RoboDK station: coursework2_ReiaMenezes_M00791121_finalsubmission.rdk

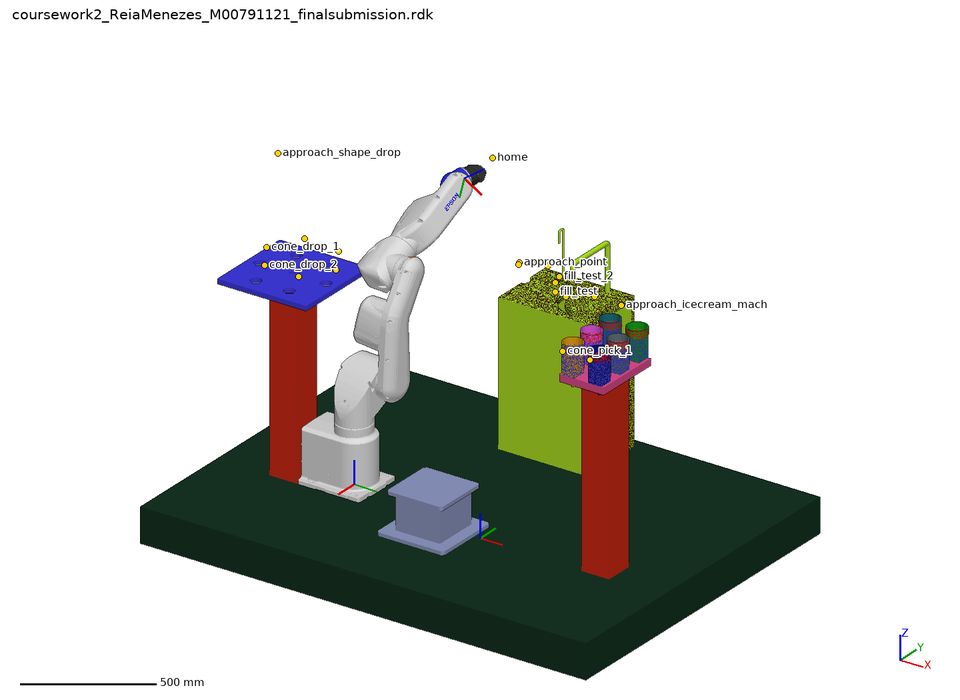
[picture v0: the station drawn from its stored meshes, robots at their saved joint values, targets as dots, program paths as lines]
Station coursework2_ReiaMenezes_M00791121_finalsubmission (saved by RoboDK 5.8.0). Poses are relative to the parent item; angles as X-Y-Z fixed-axis rotations.
Station parameters (name, value as stored): 153.91
  - frame Base_cell_frame at (0, 0, 0) mm
    - object PDE4431_CW2_2024 at (0, 0, 0) mm, rotated rx 90 ry 0 rz 0 deg, size 2000 x 980 x 1500 mm, geometry from PDE4431_CW2_2024.STEP
    - frame Epson VT6 Base at (-250, -450, 330) mm, rotated rx 0 ry 0 rz -90 deg
      - robot Epson VT6: 6 axes, payload 6 kg, reach 920 mm, repeatability 0.1 mm, weight 40 kg
          modified DH rows (alpha deg, a mm, theta deg, d mm): 0, 0, 0, 412; -90, 100, -90, 0; 0, 420, 0, 0; -90, 0, 0, 400; 90, 0, 0, 0; -90, 0, 0, 80
          base shift (0, 0, 0) mm, rotated rx 0 ry 0 rz 90 deg
          joint limits [-170, -160, -51, -200, -125, -360] to [170, 65, 190, 200, 125, 360]; home [0, 0, 0, 0, 0, 0]; saved at [85.974, -13.175, 41.561, 23.33, -25.202, -130.293]
        - frame RobotiQ 2F-140 Gripper (Mechanism) Base at (0, 0, 0) mm
          - robot RobotiQ 2F-140 Gripper (Mechanism) (model RobotiQ 2F140): 1 axes, payload 5 kg
              joint limits [0] to [140]; home [140]; saved at [99.47]
          - target open_gripper (Cartesian target) at (0, 0, 135) mm, rotated rx -90 ry 0 rz 90 deg; joints [99.47, 14.65, 163.72, -0.95, 89.45, -5.12] of RobotiQ 2F-140 Gripper (Mechanism)
          - target close_gripper (Cartesian target) at (0, 0, 135) mm, rotated rx -90 ry 0 rz 90 deg; joints [60, 27.47, -32.86, -122.29, -24.8, -148.93] of RobotiQ 2F-140 Gripper (Mechanism)
        - tool Tool 1, TCP at (-20, -10, 155) mm, rotated rx -100 ry 0 rz 70 deg
    - object Pedestal_1 at (0, -300, 150) mm, rotated rx 90 ry 0 rz 0 deg, size 300 x 180 x 300 mm, geometry from Pedestal_1.STEP
    - frame input_table_frame at (0, 0, 0) mm
      - target home (Cartesian target) at (-171.13, 326, 1377.48) mm, rotated rx -102.04 ry 85.05 rz 74.18 deg; joints [82.41, -18.36, 51.51, -8.06, -28.54, -82.2] of Epson VT6
      - target approach_point (Cartesian target) at (397.26, -315.09, 1365.72) mm, rotated rx -100.11 ry -87.63 rz -171.58 deg; joints [18.089, -0.789, 29.967, 38.658, -32.785, 56.501] of Epson VT6
      - target cone_pick_1 (Cartesian target) at (594.91, -318.66, 1058.51) mm, rotated rx -100.11 ry -87.63 rz -171.58 deg; joints [7.923, -20.29, 7.849, 146.461, -17.595, -57.734] of Epson VT6
      - target cone_pick_2 (Cartesian target) at (715.78, -319.07, 1058.49) mm, rotated rx -126.16 ry -87.1 rz -145.13 deg; joints [6.525, -37.672, 34.127, 126.782, -9.811, -38.578] of Epson VT6
      - target approach_icecream_machine_point (Cartesian target) at (301.22, 477.28, 847.78) mm, rotated rx -50.46 ry -87.49 rz -131.29 deg; joints [-33.96, -23.408, -22.424, 40.243, 55.613, 64.831] of Epson VT6
      - target starting_icecream (Cartesian target) at (181.46, 475.85, 849.63) mm, rotated rx -100.83 ry -88.03 rz -80.88 deg; joints [59.132, -56.563, 37.437, 56.856, 35.551, 37.301] of Epson VT6
      - target fill_down_flavor1 (Cartesian target) at (99.43, 408.13, 852.78) mm, rotated rx -100.83 ry -88.03 rz -80.88 deg; joints [61.936, -42.802, 12.032, 42.314, 41.214, 54.267] of Epson VT6
      - target fill_test (Cartesian target) at (39.88, 425.07, 848.67) mm, rotated rx -100.83 ry -88.03 rz -80.88 deg; joints [66.768, -41.855, 9.609, 34.939, 39.793, 60.64] of Epson VT6
      - target approach_icecream_2 (Cartesian target) at (-3.3, 486.34, 850.99) mm, rotated rx -100.83 ry -88.03 rz -80.88 deg; joints [71.584, -46.813, 19.15, 31.191, 33.677, 62.31] of Epson VT6
      - target fill_down_flavor2 (Cartesian target) at (-100.56, 579.23, 854.68) mm, rotated rx -100.83 ry -88.03 rz -80.88 deg; joints [79.404, -48.826, 23.503, 18.809, 28.583, 72.676] of Epson VT6
      - target fill_test_icecream (Cartesian target) at (-140.12, 595.57, 850.44) mm, rotated rx -100.83 ry -88.03 rz -80.88 deg; joints [82.903, -57.981, 40.297, 15.654, 20.323, 74.725] of Epson VT6
      - target fill_test_3 (Cartesian target) at (-161.01, 566.2, 849.56) mm, rotated rx -100.83 ry -88.03 rz -80.88 deg; joints [84.119, -53.062, 30.713, 10.031, 24.622, 80.354] of Epson VT6
      - target completed_icecream_machine (Cartesian target) at (-201.89, 537.42, 848.81) mm, rotated rx -100.83 ry -88.03 rz -80.88 deg; joints [86.913, -48.679, 22.293, 2.884, 28.353, 87.045] of Epson VT6
      - target approach_shape_drop (Cartesian target) at (-801.01, -152.39, 1410.63) mm, rotated rx -121.97 ry -88.27 rz 29.1 deg; joints [139.545, -3.407, 40.97, 127.197, 49.933, -51.748] of Epson VT6
      - target cone_drop_1 (Cartesian target) at (-813.15, -207.69, 1046.6) mm, rotated rx -121.97 ry -88.27 rz 29.1 deg; joints [152.488, 12.57, -28.659, 56.431, 30.004, 35.87] of Epson VT6
      - target cone_drop_2 (Cartesian target) at (-731.62, -336.84, 1047.6) mm, rotated rx -102.73 ry -87.66 rz 14.29 deg; joints [155.972, 28.648, -38.95, 65.094, 28.402, 26.221] of Epson VT6
      - target cone_drop_3 (Cartesian target) at (-739.03, -66.95, 1045.18) mm, rotated rx -102.73 ry -87.66 rz 14.29 deg; joints [125.197, 0.545, -18.808, 75.749, 59.119, 22.393] of Epson VT6
      - target cone_drop_4 (Cartesian target) at (-581.8, -332.78, 1041.64) mm, rotated rx -102.73 ry -87.66 rz 14.29 deg; joints [133.571, 51.579, -47.266, 90.821, 47.936, -4.268] of Epson VT6
      - target cone_drop_5 (Cartesian target) at (-583.93, -72.76, 1039.1) mm, rotated rx -102.73 ry -87.66 rz 14.29 deg; joints [107.283, 10.862, -28.91, 82.785, 75.803, 18.747] of Epson VT6
      - target cone_drop_6 (Cartesian target) at (-505.45, -200.67, 1037.29) mm, rotated rx -102.73 ry -87.66 rz 14.29 deg; joints [99.064, 34.372, -42.989, 86.597, 82.923, 8.461] of Epson VT6
      - target fill_test_2 (Cartesian target) at (-16.95, 531.74, 852.61) mm, rotated rx -100.83 ry -88.03 rz -80.88 deg; joints [73.539, -52.018, 29.199, 32.068, 28.624, 60.312] of Epson VT6
      - target fill_test_4 (Cartesian target) at (166.07, 460.97, 859.21) mm, rotated rx -100.83 ry -88.03 rz -80.88 deg; joints [59.527, -52.804, 31.711, 54.194, 36.359, 40.421] of Epson VT6
      - object Cone_2 at (760, -320, 1030) mm, rotated rx 90 ry 0 rz 0 deg, size 84.9 x 182 x 85 mm, geometry from Cone-Part.STEP
      - object Cone_1 at (640, -320, 1030) mm, rotated rx 90 ry 0 rz 0 deg, size 84.9 x 182 x 85 mm, geometry from Cone-Part.STEP
      - object Cone_3 at (640, -200, 1030) mm, rotated rx 90 ry 0 rz 0 deg, size 84.9 x 182 x 85 mm, geometry from Cone-Part.STEP
      - object Cone_4 at (760, -200, 1030) mm, rotated rx 90 ry 0 rz 0 deg, size 84.9 x 182 x 85 mm, geometry from Cone-Part.STEP
      - object Cone_5 at (640, -80, 1030) mm, rotated rx 90 ry 0 rz 0 deg, size 84.9 x 182 x 85 mm, geometry from Cone-Part.STEP
      - object Cone_6 at (760, -80, 1030) mm, rotated rx 90 ry 0 rz 0 deg, size 84.9 x 182 x 85 mm, geometry from Cone-Part.STEP
  - Python program icecream_filling_process (listed below)
  - program open_gripper_mechanism (2 instructions, listed below)
  - program close_gripper_mechanism (2 instructions, listed below)
  - program attach_cone (1 instructions, listed below)
  - program detach_cone (1 instructions, listed below)
  - program replace_cone1 (1 instructions, listed below)
  - program replace_cone2 (1 instructions, listed below)
  - program replace_cone3 (1 instructions, listed below)
  - program replace_cone4 (1 instructions, listed below)
  - program replace_cone5 (1 instructions, listed below)
  - program replace_cone6 (1 instructions, listed below)

--- Python program icecream_filling_process ---
from robodk import *
from robodk.robolink import *
from robodk.robomath import *
import time

# creating a connection to robodk
RDK = Robolink()
robot = RDK.Item('Epson VT6')

# programs for gripper operations - opening and closing
open_gripper_mechanism_program = RDK.Item('open_gripper_mechanism', ITEM_TYPE_PROGRAM)
close_gripper_mechanism_program = RDK.Item('close_gripper_mechanism', ITEM_TYPE_PROGRAM)
attach_cone = RDK.Item('attach_cone', ITEM_TYPE_PROGRAM)
detach_cone = RDK.Item('detach_cone', ITEM_TYPE_PROGRAM)
home = RDK.Item('home')  # home position of the robot

# define positions for picking the cones from the first station
cone_pick_1 = RDK.Item('cone_pick_1')  # first cone position
cone_pick_2 = RDK.Item('cone_pick_2')  # second cone position
cone_pick_3 = cone_pick_1.Pose() * transl(0, 0, -120)  # third cone position
cone_pick_4 = cone_pick_2.Pose() * transl(0, 0, -120)  # fourth cone position
cone_pick_5 = cone_pick_1.Pose() * transl(0, 0, -240)  # fifth cone position
cone_pick_6 = cone_pick_2.Pose() * transl(0, 0, -240)  # sixth cone position
approach_point = RDK.Item('approach_point')  # approach position for picking cones from the first station

# define positions for ice cream filling
approach_icecream_machine_point = RDK.Item('approach_icecream_machine_point')  # approach to ice cream machine
starting_icecream = RDK.Item('starting_icecream')  # initial ice cream machine position
fill_down_flavor1 = RDK.Item('fill_down_flavor1')  # position for first flavor filling
fill_down_flavor2 = RDK.Item('fill_down_flavor2')  # position for second flavor filling

# define fill positions with downward and upward transformations
fill_1_go_down = fill_down_flavor1.Pose() * transl(0, 0, -30)  # move down for first flavor
fill_1_go_up = fill_1_go_down * transl(0, 0, 30)  # move back up for first flavor
fill_2_go_down = fill_down_flavor2.Pose() * transl(0, 0, -30)  # move down for second flavor
fill_2_go_up = fill_2_go_down * transl(0, 0, 30)  # move back up for second flavor
completed_icecream_machine = RDK.Item('completed_icecream_machine')  # final position at ice cream machine - completed

# define positions for dropping cones
cone_drop_1 = RDK.Item('cone_drop_1')  # first cone drop position
cone_drop_2 = RDK.Item('cone_drop_2')  # second cone drop position
cone_drop_3 = RDK.Item('cone_drop_3')  # third cone drop position
cone_drop_4 = RDK.Item('cone_drop_4')  # fourth cone drop position
cone_drop_5 = RDK.Item('cone_drop_5')  # fifth cone drop position
cone_drop_6 = RDK.Item('cone_drop_6')  # sixth cone drop position

# define approach drop positions with adjusted transformations
approach_drop_cone1 = cone_drop_1.Pose() * transl(-50, 0, 50)  # approach position for cone 1 drop
approach_drop_cone2 = cone_drop_2.Pose() * transl(-50, 0, 50)  # approach position for cone 2 drop
approach_drop_cone3 = cone_drop_3.Pose() * transl(-50, 0, 50)  # approach position for cone 3 drop
approach_drop_cone4 = cone_drop_4.Pose() * transl(-20, 0, 20)  # approach position for cone 4 drop (adjusted) - too close for the robot target reach
approach_drop_cone5 = cone_drop_5.Pose() * transl(-50, 0, 50)  # approach position for cone 5 drop
approach_drop_cone6 = cone_drop_6.Pose() * transl(-50, 0, 50)  # approach position for cone 6 drop

# create arrays for cone positions
pick_cone_positions = [cone_pick_1, cone_pick_2, cone_pick_3, cone_pick_4, cone_pick_5, cone_pick_6]
approach_cone_drop_positions = [approach_drop_cone1, approach_drop_cone2, approach_drop_cone3, approach_drop_cone4, approach_drop_cone5, approach_drop_cone6]
drop_cone_positions = [cone_drop_1, cone_drop_2, cone_drop_3, cone_drop_4, cone_drop_5, cone_drop_6]

# created a loop for picking, filling, and dropping cones
for i in range(6):
    try:
        print(f"starting sequence for cone {i+1}")
        robot.MoveJ(home)  # move to home position
        open_gripper_mechanism_program.RunProgram()  # open gripper
        robot.MoveJ(approach_point)  # move to approach point
        robot.MoveL(pick_cone_positions[i])  # move to pick position
        close_gripper_mechanism_program.RunProgram()  # close gripper
        attach_cone.RunProgram()  # attach cone to gripper
        robot.MoveL(approach_point)  # return to approach point
        robot.MoveJ(approach_icecream_machine_point)  # move to ice cream machine
        robot.MoveL(starting_icecream)  # move to starting position at machine

        # filling process
        robot.setSpeed(50)  # set slower speed for filling
        robot.setSpeedJoints(25)
        robot.MoveL(fill_down_flavor1)  # move to first flavor position
        robot.MoveL(fill_1_go_down)  # move down to fill
        robot.MoveL(fill_1_go_up)  # move up after filling
        robot.MoveL(fill_down_flavor2)  # move to second flavor position
        robot.MoveL(fill_2_go_down)  # move down to fill
        robot.MoveL(fill_2_go_up)  # move up after filling
        robot.MoveL(completed_icecream_machine)  # move to completed position
        robot.setSpeed(500)  # restore normal speed
        robot.setSpeedJoints(150)

        # dropping process
        print(f"dropping cone {i+1}")
        robot.MoveL(approach_cone_drop_positions[i])  # move to approach drop position
        robot.MoveL(drop_cone_positions[i])  # move to drop position
        detach_cone.RunProgram()  # detach cone from gripper
        open_gripper_mechanism_program.RunProgram()  # open gripper
        robot.MoveL(approach_cone_drop_positions[i])  # return to approach drop position
    except Exception as e:
        print(f"error during sequence for cone {i+1}: {e}")
        continue

# return to home position
print("all cones have been filled with ice cream. returning the robot to home position.")
robot.MoveJ(home)

--- program open_gripper_mechanism (robot RobotiQ 2F-140 Gripper (Mechanism)) ---
  Set Ref.: RobotiQ 2F-140 Gripper (Mechanism) Base
  MoveJ (open_gripper)

--- program close_gripper_mechanism (robot RobotiQ 2F-140 Gripper (Mechanism)) ---
  Set Ref.: RobotiQ 2F-140 Gripper (Mechanism) Base
  MoveJ (close_gripper)

--- program attach_cone (robot Epson VT6) ---
  Attach to Tool 1

--- program detach_cone (robot Epson VT6) ---
  Detach from Tool 1

--- program replace_cone1 (robot Epson VT6) ---
  Replace objects

--- program replace_cone2 (robot Epson VT6) ---
  Replace objects

--- program replace_cone3 (robot Epson VT6) ---
  Replace objects

--- program replace_cone4 (robot Epson VT6) ---
  Replace objects

--- program replace_cone5 (robot Epson VT6) ---
  Replace objects

--- program replace_cone6 (robot Epson VT6) ---
  Replace objects
